FUNCTION TryConvert_SINT_TO_INT : BOOL
VAR_INPUT
	in : SINT;
	out : REFERENCE TO INT;
END_VAR

out := SINT_TO_INT(in);
TryConvert_SINT_TO_INT := TRUE;

END_FUNCTION

(* stored: Version 1.1.0.1, ProductVersion 3.1.4024.12
   POU TryConvert_SINT_TO_INT: Id {e6374bfe-3695-4092-8131-00217969486a}, SpecialFunc None *)
